{attribute addProperty BoxType "EL9221-4030-0018"}
{attribute addProperty Id "StatusAT %I*Status_EBB67327324"}
{attribute addProperty CRC "4261982012"}
{attribute addProperty SizeInBites "32"}
{attribute addProperty SizeInBytes "4"}
TYPE OCP_Inputs_FE08AF3C :
STRUCT
	{attribute addProperty Name "Status"}
	Status AT %I* : Status_EBB67327;
END_STRUCT
END_TYPE

(* stored: Version 1.2.0.0, ProductVersion 3.1.4024.9
   DUT OCP_Inputs_FE08AF3C: Id {cf6ba5f6-2792-4a76-bb2e-e40f71e42cd2} *)
